{attribute 'TcGenerated'}
{attribute 'no-analysis'}
{attribute 'linkalways'}
// This function has been automatically generated from the project information.
VAR_GLOBAL CONSTANT
    {attribute 'const_non_replaced'}
    stLibVersion_lcls_twincat_motion : ST_LibVersion := (iMajor := 4, iMinor := 5, iBuild := 1, iRevision := 0, nFlags := 1, sVersion := '4.5.1');
END_VAR

(* stored: Version 1.1.0.1
   GVL Global_Version: Id {48ba44b1-4c68-4b26-a068-30d566aa0387} *)
